FUNCTION GetTick : UDINT
VAR_INPUT
END_VAR
VAR
END_VAR

GetTick := TO_UDINT(F_GetTaskTime()/10000);

END_FUNCTION

(* stored: Version 1.1.0.1, ProductVersion 3.1.4024.6
   POU GetTick: Id {29921add-6e89-4945-967a-5cd442b28ed3}, SpecialFunc None *)
